// ---- Modules/12 FG_02/FG_02.TcPOU
// FG_02 - optical inspection. Camera handshake, no moving parts.
// Triggered by Index02; reports OperationDone. A NOK aborts (fault 1).
// Twin side: FB_Camera in OC_SIM - both halves must agree on the bit layout,
// and nothing checks it for you.
// Contract: _workflow/reference/fg-02-behaviour.md
FUNCTION_BLOCK FG_02 EXTENDS FB_PackML_BaseModule
VAR
	P_Camera	: FB_AbstractCamera := (Name := 'P_Camera');

	// Group level fault - see ST_FG_02_Inspection_Status. Cleared in Clearing.
	_FaultCode		: DINT;
	// The verdict of the last completed shot, latched so the panel still shows it
	// once ResultValid has dropped.
	_LastResultOK	: BOOL;

	{ attribute 'TcHmiSymbol.AddSymbol' }
	HMI : ST_HMI_FG_02;
END_VAR

METHOD PROTECTED Aborting
VAR_INPUT
END_VAR
// Disable() drops the trigger before the enable, so a shot is never left armed.
CASE SequenceState OF
	0:
		NoStateTasksToComplete	:= FALSE;
		P_Camera.Disable();
		SequenceState			:= SequenceState + 10;

	10:
		StateTasksComplete := TRUE;
END_CASE

SUPER^.Aborting();
END_METHOD

METHOD PROTECTED Clearing
VAR_INPUT
END_VAR
CASE SequenceState OF
	0:
		NoStateTasksToComplete := FALSE;
		// Cleared by the act of clearing, not by the condition going away.
		_FaultCode := 0;
		SequenceState := SequenceState + 10;

	10:	// Clear any latched component alarm.
		IF P_Camera.Reset() THEN
			SequenceState := SequenceState + 10;
		END_IF

	20:
		StateTasksComplete := TRUE;
END_CASE

SUPER^.Clearing();
END_METHOD

METHOD PUBLIC CyclicLogic
VAR_INPUT
END_VAR
IF NOT _InitComplete THEN
	_InitComplete := Initialize();
	RETURN;
END_IF

// No process image copy step: component members map straight to terminal channels.
SUPER^.CyclicLogic();

PublishStatus();
END_METHOD

METHOD PROTECTED Execute
VAR_INPUT
END_VAR
VAR_INST
	ReadyTimer	: TON;
	ShotTimer	: TON;
END_VAR
// The vision-sensor handshake. Every wait is bounded; every timeout faults.

CASE _CurrentMode OF

	//============================= PRODUCTION =================================
	E_PMLUnitMode.ePMLUnitMode_Production:

		CASE SequenceState OF
			0:
				NoStateTasksToComplete	:= FALSE;
				P_Camera.Disable();
				SequenceState			:= SequenceState + 10;

			10:	// Power up, wait for Ready. Timeout -> the camera is not answering.
				P_Camera.Enable();
				IF P_Camera.Ready THEN
					SequenceState := SequenceState + 10;
				ELSIF ReadyTimer.Q THEN
					_FaultCode := 2;
					AbortImmediate();
				END_IF

			20:	// Trigger. ResultValid also acknowledges: a fast camera can raise
				// and drop Busy inside one scan.
				P_Camera.Trigger();
				IF P_Camera.DeviceBusy OR P_Camera.ResultValid THEN
					SequenceState := SequenceState + 10;
				ELSIF ShotTimer.Q THEN
					_FaultCode := 3;
					AbortImmediate();
				END_IF

			30:	// Read the verdict. It stands until the trigger is released.
				IF P_Camera.ResultValid THEN
					_LastResultOK := P_Camera.ResultOK;
					IF P_Camera.ResultOK THEN
						SequenceState := SequenceState + 10;
					ELSE
						_FaultCode := 1;
						AbortImmediate();
					END_IF
				ELSIF ShotTimer.Q THEN
					_FaultCode := 3;
					AbortImmediate();
				END_IF

			40:	// Power down. Disable() clears the trigger first, which tells the
				// camera its verdict was read.
				P_Camera.Disable();
				SequenceState := SequenceState + 10;

			50:	// Execute is the one acting state that does not self-complete.
				// StateComplete() would be wrong here.
				ChangeState(E_PMLCommand.ePMLCommand_Complete);
		END_CASE

	//======================= MAINTENANCE & MANUAL =============================
	E_PMLUnitMode.ePMLUnitMode_Maintenance, E_PMLUnitMode.ePMLUnitMode_Manual:
		// No group sequence. The camera stays reachable through its own
		// component HMI control.
		;
END_CASE

SUPER^.Execute();

// ShotTimer spans steps 20 and 30 on purpose: the camera's total response time is
// one number, and that is what an operator is told.
ReadyTimer(IN := SequenceState = 10,								PT := T#2S);
ShotTimer(IN := (SequenceState = 20) OR (SequenceState = 30),		PT := T#3S);
END_METHOD

METHOD PROTECTED HMICommunication
VAR_INPUT
END_VAR
// Command half of the HMI bridge; PublishStatus is the status half. MUST be in
// this method: the base calls it immediately before ModeControl() and
// StateControl(), and reads its own PackMLBaseModule_HMI.Command, never ours.
PackMLBaseModule_HMI.Command := HMI.Command;

SUPER^.HMICommunication();

// The base clears a latch by writing back the value it acted on.
HMI.Command := PackMLBaseModule_HMI.Command;
END_METHOD

METHOD PROTECTED Initialize : BOOL;
VAR
END_VAR
Initialize := FALSE;

CASE DescendantSequenceState OF
	0:
		RegisterComponent(P_Camera);

		_LogModeChanges		:= FALSE;
		_LogStateChanges	:= TRUE;
		HMI.Config.Name		:= THIS^._Name;
		DescendantSequenceState := DescendantSequenceState + 10;

	10:
		// No travel timeouts - nothing in this group moves.
		DescendantSequenceState := DescendantSequenceState + 10;

	20:
		IF SUPER^.Initialize() THEN
			DescendantSequenceState := DescendantSequenceState + 10;
		END_IF

	30:
		Initialize := TRUE;
END_CASE
END_METHOD

ACTION PublishStatus:
// Status half of the HMI bridge. Called AFTER SUPER^.CyclicLogic(), so every
// field is this scan's. Copy the base struct wholesale - setting fields one by one
// leaves Busy, Error, ErrorID and HMIControlAvailable at zero.
// P_Camera publishes its own handshake; what is added here is what no device owns.
HMI.Config		:= PackMLBaseModule_HMI.Config;
HMI.Status		:= PackMLBaseModule_HMI.Status;

HMI.StateName				:= F_PMLStateName(_CurrentState);
HMI.Sequence.StepIndex		:= SequenceState;
HMI.Inspection.FaultCode	:= _FaultCode;
HMI.Inspection.LastResultOK	:= _LastResultOK;
END_ACTION

METHOD PROTECTED Resetting
VAR_INPUT
END_VAR
// Home is "nothing energised". Terminates on its own call and nothing else.

CASE SequenceState OF
	0:
		NoStateTasksToComplete	:= FALSE;
		P_Camera.Disable();
		SequenceState			:= SequenceState + 10;

	10:
		StateTasksComplete := TRUE;
END_CASE

SUPER^.Resetting();
END_METHOD

METHOD PROTECTED Stopping
VAR_INPUT
END_VAR
CASE SequenceState OF
	0:
		NoStateTasksToComplete	:= FALSE;
		P_Camera.Disable();
		SequenceState			:= SequenceState + 10;

	10:
		StateTasksComplete := TRUE;
END_CASE

SUPER^.Stopping();
END_METHOD

END_FUNCTION_BLOCK

// ---- Modules/13 FG_03/FG_03.TcPOU
// FG_03 - slot 1 to slot 2 transfer, with a 180 degree flip.
// !! THE TWO ARMS NAME THEIR AXES THE OPPOSITE WAY ROUND. Arm 1: X1 vertical,
// Y1 horizontal. Arm 2: X2 horizontal, Y2 vertical (factor -0.001, so a rising
// value descends). Every earlier version of this file had arm 1 wrong.
// Arm 1 NEVER lowers to place - the R1 flip is what carries the part down.
// A cylinder limit is not a grip witness: only B_Detect1/B_Detect2 are.
// Contract: _workflow/reference/fg-03-behaviour.md and gripper-station-reset.md
FUNCTION_BLOCK FG_03 EXTENDS FB_PackML_BaseModule
VAR
	// --- Arm 1, the placing arm ---------------------------------------------
	{ attribute 'TcHmiSymbol.AddSymbol' }
	Y_AxisX1	: FB_DoubleSolenoidFeedback := (Name := 'Y_AxisX1');
	{ attribute 'TcHmiSymbol.AddSymbol' }
	Y_AxisY1	: FB_DoubleSolenoidFeedback := (Name := 'Y_AxisY1');
	{ attribute 'TcHmiSymbol.AddSymbol' }
	Y_AxisR1	: FB_DoubleSolenoidFeedback := (Name := 'Y_AxisR1');
	{ attribute 'TcHmiSymbol.AddSymbol' }
	Y_Gripper1	: FB_DoubleSolenoidFeedback := (Name := 'Y_Gripper1');
	{ attribute 'TcHmiSymbol.AddSymbol' }
	B_Detect1	: FB_DigitalSensor := (Name := 'B_Detect1');

	// --- Arm 2, the picking arm ---------------------------------------------
	{ attribute 'TcHmiSymbol.AddSymbol' }
	Y_AxisX2	: FB_DoubleSolenoidFeedback := (Name := 'Y_AxisX2');
	{ attribute 'TcHmiSymbol.AddSymbol' }
	Y_AxisY2	: FB_DoubleSolenoidFeedback := (Name := 'Y_AxisY2');
	{ attribute 'TcHmiSymbol.AddSymbol' }
	Y_Gripper2	: FB_DoubleSolenoidFeedback := (Name := 'Y_Gripper2');
	{ attribute 'TcHmiSymbol.AddSymbol' }
	B_Detect2	: FB_DigitalSensor := (Name := 'B_Detect2');

	// Group level fault - see ST_FG_03_Transfer_Status. Cleared in Clearing.
	_FaultCode	: DINT;

	// What Resetting found in the grippers, sampled ONCE at its step 0. They decide
	// which grippers it may open and which way it turns arm 1, and the fact that they
	// are a snapshot rather than a live read is the whole reason the reset cannot
	// hang: no step waits on a sensor, only on its own cylinders. Step 10 clears
	// _Held2 when it has VERIFIED arm 2 let go - updating the snapshot from a checked
	// fact, which is not the same thing as reading the sensor in a wait.
	_Held1		: BOOL;
	_Held2		: BOOL;

	{ attribute 'TcHmiSymbol.AddSymbol' }
	HMI : ST_HMI_FG_03;
END_VAR

METHOD PROTECTED Aborting
VAR_INPUT
END_VAR
// AN ABORT COMMANDS NO MOTION IN THIS GROUP, and that is the whole design.
// No hazardous output to kill. What there is, at almost every step, is a part held
// in the air, and commanding an axis on an abort risks dropping it.
// COMMANDING NOTHING IS NOT THE SAME AS HOLDING ON: the grippers are held closed
// by the CyclicLogic interlock. This method leaves the AXES alone.
// Homing happens in Resetting, where the operator has asked for it.
CASE SequenceState OF
	0:
		NoStateTasksToComplete	:= FALSE;
		SequenceState			:= SequenceState + 10;

	10:
		StateTasksComplete := TRUE;
END_CASE

SUPER^.Aborting();
END_METHOD

METHOD PROTECTED Clearing
VAR_INPUT
END_VAR
CASE SequenceState OF
	0:
		NoStateTasksToComplete := FALSE;
		// The group fault is cleared by the act of clearing, not by the condition
		// going away. A part jammed in a gripper is still jammed after the sensor
		// has stopped being interesting; the operator has to have taken it out, and
		// Execute's step 0 guard is what checks that they did.
		_FaultCode := 0;
		SequenceState := SequenceState + 10;

	10:	// Clear latched component alarms - the solenoid travel timeouts latch.
		IF Y_AxisX1.Reset()
			AND Y_AxisY1.Reset()
			AND Y_AxisR1.Reset()
			AND Y_Gripper1.Reset()
			AND B_Detect1.Reset()
			AND Y_AxisX2.Reset()
			AND Y_AxisY2.Reset()
			AND Y_Gripper2.Reset()
			AND B_Detect2.Reset() THEN
			SequenceState := SequenceState + 10;
		END_IF

	20:
		StateTasksComplete := TRUE;
END_CASE

SUPER^.Clearing();
END_METHOD

METHOD PUBLIC CyclicLogic
VAR_INPUT
END_VAR
IF NOT _InitComplete THEN
	_InitComplete := Initialize();
	RETURN;
END_IF

// A HELD PART IS GRIPPED ACTIVELY, IN EVERY STATE EXCEPT Execute.
//
// A DE-ENERGISED DOUBLE SOLENOID DOES NOT HOLD THE PART IN THE TWIN. True of the
// real valve, false here. The scene wires the gripper cylinder as:
//     OnLimitMaxEvent  -> Gripper.Pick(bool)
//     OnLimitMinEvent  -> Gripper.Place(bool)
//     OnActiveChanged  -> Gripper.Place(bool)    IsActive = "moving"
// and Cylinder sets IsActive := (target <> value), so the payload is held only
// while the cylinder is at max AND STANDING STILL. Leaving it uncommanded through
// Clearing and Resetting was enough to nudge it off the limit, and arm 1 dropped
// its part mid-reset.
//
// So the grip is re-asserted every scan off the live sensor. It commands no MOTION
// - Extend on a closed gripper is a no-op at the valve.
// BEFORE SUPER^, WHICH IS WHAT MAKES IT AN INTERLOCK: it overwrites whatever a
// state method asked for on the previous scan. HMICommunication runs inside SUPER^
// and still gets the last word, so Manual can jog a gripper open.
// Execute is excluded because Execute is the only state allowed to put a part down.
IF _CurrentState <> E_PMLState.ePMLState_Execute THEN
	IF B_Detect1.Active THEN
		Y_Gripper1.Extend();
	END_IF
	IF B_Detect2.Active THEN
		Y_Gripper2.Extend();
	END_IF
END_IF

// No process image copy step: component process-image members are mapped directly
// to terminal channels.
SUPER^.CyclicLogic();

PublishStatus();
END_METHOD

METHOD PROTECTED Execute
VAR_INPUT
END_VAR
VAR_INST
	SettleTimer		: TON;

	// One grace timer per confirming step, and they cannot be shared. Steps 90 and
	// 100 are adjacent, so a timer armed on "either of them" would never see its IN
	// drop between the two and would carry step 80's elapsed time into step 90.
	// Each is armed only once its cylinder has reached its limit: the cylinder's own
	// ExtendTime/RetractTime covers the travel, and this covers only the question
	// that follows it - did the payload do what the stroke was supposed to make it do.
	PickTimer		: TON;
	HandoverTimer	: TON;
	Release2Timer	: TON;
	Release1Timer	: TON;
END_VAR
// Ordering from the authored Process entry, confirmed motion by motion against
// The SIL's 0.2 s dwells are replaced by the limit switches they stood in for.
// EVERY GRIP AND EVERY RELEASE IS CONFIRMED BY A SENSOR, not by the cylinder limit
// alone: a gripper closing on nothing reaches Extended SOONER than one closing on
// a part, so .Extended proves the jaws moved, never that they caught anything.
// Each confirmation is bounded and faults rather than waiting; the cylinder's own
// travel timeout covers the stroke, these timers only the question after it.

CASE _CurrentMode OF

	//============================= PRODUCTION =================================
	E_PMLUnitMode.ePMLUnitMode_Production:

		CASE SequenceState OF
			0:	// WHERE THE CYCLE STARTS IS DERIVED, NOT REMEMBERED. A part in a
				// gripper is a legal starting condition: Resetting parks a held part
				// at its arm's safe position instead of putting it back, so the next
				// Start picks the cycle up from there. Which sub-sequence that is
				// follows from which gripper is carrying something and from nothing
				// else - no stored step index, no "was I interrupted" flag.
				//
				// The arm must actually BE at its safe position. If a part is held
				// somewhere else - someone jogged an axis in Manual - the entry point
				// would be a guess, so this refuses rather than moves. Reset is the
				// recovery: Resetting reaches a safe position from anywhere.
				NoStateTasksToComplete	:= FALSE;

				IF B_Detect1.Active THEN
					IF Y_AxisX1.Extended AND Y_AxisY1.Retracted AND Y_AxisR1.Retracted THEN
						SequenceState := 100;		// at SAFE B - resume into SUB 3
					ELSE
						_FaultCode := 5;
						AbortImmediate();
					END_IF

				ELSIF B_Detect2.Active THEN
					IF Y_AxisX2.Retracted AND Y_AxisY2.Retracted THEN
						SequenceState := 50;		// at SAFE A - resume into SUB 2
					ELSE
						_FaultCode := 5;
						AbortImmediate();
					END_IF

				ELSE
					SequenceState := 10;			// nothing held - the whole cycle
				END_IF

			10:	// Let the pallet settle on the index lift before touching it. No
				// sensor reports this, so it is a timer. A resume skips this step
				// entirely - the pallet has been standing still since the E-Stop.
				IF SettleTimer.Q THEN
					SequenceState := SequenceState + 10;
				END_IF

		//===================== SUB 1 - pick out of slot 1 ======================
		// Entered only with both grippers empty. Ends at SAFE A.
			20:	// Arm 2 down into slot 1. Arm in Ready pos
				Y_AxisX1.Extend();
				Y_AxisY2.Extend();
				IF Y_AxisY2.Extended THEN
					SequenceState := SequenceState + 10;
				END_IF
				

			30:	// Grip the part, and confirm the grip caught something. An empty
				// slot 1, a mispositioned pallet or a part that slipped all look
				// identical on the cylinder limit and are all fault 2 here.
				Y_Gripper2.Extend();
				IF Y_Gripper2.Extended THEN
					IF B_Detect2.Active THEN
						SequenceState := SequenceState + 10;
					ELSIF PickTimer.Q THEN
						_FaultCode := 2;
						AbortImmediate();
					END_IF
				END_IF

			40:	// Lift clear of the pallet before anything traverses.
				//
				// *** SAFE A *** - X2 min, Y2 min, part in gripper 2. Arm 2 raised at
				// its home over slot 1. This is a state the cycle passes through in
				// the ordinary course, which is why a resume re-enters at step 50 and
				// nothing had to be inserted to make the position real.
				Y_AxisY2.Retract();
				IF Y_AxisY2.Retracted THEN
					SequenceState := SequenceState + 10;
				END_IF

		//=================== SUB 2 - the transfer (resume: 50) =================
		// Entered with the part in gripper 2 and arm 2 at SAFE A. Ends at SAFE B.
			50:	// Arm 2 traverses to the transfer position
				Y_AxisX2.Extend();
				IF Y_AxisX2.Extended THEN
					SequenceState := SequenceState + 10;
				END_IF

			60:	// ARM 1 RISES, AND THEN STAYS UP FOR THE WHOLE CYCLE. 			
				IF Y_AxisX1.Extended THEN
					SequenceState := SequenceState + 10;
				END_IF

			70:	// Arm 1 traverses across to meet arm 2. 
				Y_AxisY1.Extend();
				IF Y_AxisY1.Extended THEN
					SequenceState := SequenceState + 10;
				END_IF

			80:	// Arm 1 takes hold. BOTH GRIPPERS NOW HOLD THE PART, and what makes
				// the next step safe is B_Detect1 - not the cylinder limit. Arm 1's
				// jaws reach Extended whether or not the part is between them, and a
				// dwell here (which is what the SIL does) proves even less. Only the
				// sensor says arm 1 actually has it, and step 90 opens arm 2 on the
				// strength of that.
				//
				// THIS IS THE ONE WINDOW WITH NO SAFE POSITION. Neither arm can move
				// while both hold one part, which is why Resetting has to break the
				// tie here before it can park anything.
				Y_Gripper1.Extend();
				IF Y_Gripper1.Extended THEN
					IF B_Detect1.Active THEN
						SequenceState := SequenceState + 10;
					ELSIF HandoverTimer.Q THEN
						_FaultCode := 3;
						AbortImmediate();
					END_IF
				END_IF

			90:	// Arm 2 lets go. Only now, and only once the part has actually left
				// its jaws - a part still in the beam when arm 2 traverses away would
				// be dragged off arm 1.
				//
				// *** SAFE B *** - X1 max, Y1 max, R1 min, part in gripper 1. Arm 1
				// raised at the transfer position, holding the part unrotated. Like
				// SAFE A this is a state the cycle really passes through, so a resume
				// re-enters at step 100 and simply carries on.
				Y_Gripper2.Retract();
				IF Y_Gripper2.Retracted THEN
					IF NOT B_Detect2.Active THEN
						SequenceState := SequenceState + 10;
					ELSIF Release2Timer.Q THEN
						_FaultCode := 4;
						AbortImmediate();
					END_IF
				END_IF

		//================= SUB 3 - place into slot 2 (resume: 100) =============
		// Entered with the part in gripper 1 at SAFE B.
			100: // Arm 2 back home over slot 1, empty. 
				Y_AxisX2.Retract();
				IF Y_AxisX2.Retracted THEN
					SequenceState := 105;
				END_IF
				
			105: //Align arm 1 with slot
				Y_AxisY1.Extend();
				IF Y_AxisY1.Extended THEN
					SequenceState := 110;
				END_IF

			110: // THE FLIP, AND IT IS ALSO THE PLACING MOVE. 
				Y_AxisR1.Extend();
				IF Y_AxisR1.Extended THEN
					SequenceState := SequenceState + 10;
				END_IF

			120: // Traverse across to slot 2, carrying the part flipped
				Y_AxisX1.Retract();
				IF Y_AxisX1.Retracted THEN
					SequenceState := SequenceState + 10;
				END_IF

			130: // Release into slot 2. Confirm the part is out of the jaws before
				// arm 1 traverses away: a part still gripped is carried back out of
				// the pallet, and Index03 would release a pallet that looks finished
				// and is empty.
				Y_Gripper1.Retract();
				IF Y_Gripper1.Retracted THEN
					IF NOT B_Detect1.Active THEN
						SequenceState := SequenceState + 10;
					ELSIF Release1Timer.Q THEN
						_FaultCode := 4;
						AbortImmediate();
					END_IF
				END_IF

			140: // Traverse clear of the part just placed. THIS IS NOT A DETOUR: the
				// rotation home at step 150 sweeps the gripper through wherever it
				// stands, and over slot 2 that is straight through the part. Arm 1
				// has to be back at the transfer position before it may turn.
				Y_AxisX1.Extend();
				IF Y_AxisX1.Extended THEN
					SequenceState := SequenceState + 10;
				END_IF

			150: // Rotate home, empty and clear
				Y_AxisR1.Retract();
				IF Y_AxisR1.Retracted THEN
					SequenceState := SequenceState + 10;
				END_IF

			160: // And back to the home position over slot 2
				Y_AxisY1.Retract();
				IF Y_AxisY1.Retracted THEN
					SequenceState := SequenceState + 10;
				END_IF

			170: // Execute is the one acting state that does not self-complete.
				// StateComplete() would be wrong here.
				ChangeState(E_PMLCommand.ePMLCommand_Complete);
		END_CASE

	//======================= MAINTENANCE & MANUAL =============================
	E_PMLUnitMode.ePMLUnitMode_Maintenance, E_PMLUnitMode.ePMLUnitMode_Manual:
		// Every cylinder is jogged through its own SolenoidHMI command struct,
		// which FB_SingleSolenoid.HMICommunication honours whenever HMIPermissions
		// has granted control. No group sequence runs and no code is needed here.
		;
END_CASE

SUPER^.Execute();

SettleTimer(IN := SequenceState = 10, PT := T#500MS);

// The payload grace timers. Each is armed only once its cylinder has reached the
// limit, so the budget is for the part settling in or falling out of the jaws, not
// for the stroke - the stroke already has ExtendTime/RetractTime on the cylinder.
// 500 ms is generous for a beam sensor that answers within one twin frame; it is
// long enough that a slow physics step cannot fault a good grip.
PickTimer(IN		:= (SequenceState = 30)  AND Y_Gripper2.Extended,	PT := T#500MS);
HandoverTimer(IN	:= (SequenceState = 80)  AND Y_Gripper1.Extended,	PT := T#500MS);
Release2Timer(IN	:= (SequenceState = 90)  AND Y_Gripper2.Retracted,	PT := T#500MS);
Release1Timer(IN	:= (SequenceState = 130) AND Y_Gripper1.Retracted,	PT := T#500MS);
END_METHOD

METHOD PROTECTED HMICommunication
VAR_INPUT
END_VAR
// The command half of the HMI bridge; PublishStatus is the status half.
//
// The base reads its OWN PackMLBaseModule_HMI.Command and never looks at ours, so
// without this a mode or state button on the FG_03 tile writes into a struct
// nothing consumes. It has to happen in this method because the base calls it
// immediately before ModeControl() and StateControl().
PackMLBaseModule_HMI.Command := HMI.Command;

SUPER^.HMICommunication();

// The base clears a latch by writing back the value it acted on, so the panel
// sees its request consumed instead of re-issuing it next scan.
HMI.Command := PackMLBaseModule_HMI.Command;
END_METHOD

METHOD PROTECTED Initialize : BOOL;
VAR
END_VAR
Initialize := FALSE;

CASE DescendantSequenceState OF
	0:
		RegisterComponent(Y_AxisX1);
		RegisterComponent(Y_AxisY1);
		RegisterComponent(Y_AxisR1);
		RegisterComponent(Y_Gripper1);
		RegisterComponent(B_Detect1);
		RegisterComponent(Y_AxisX2);
		RegisterComponent(Y_AxisY2);
		RegisterComponent(Y_Gripper2);
		RegisterComponent(B_Detect2);

		_LogModeChanges		:= FALSE;
		_LogStateChanges	:= TRUE;
		HMI.Config.Name		:= THIS^._Name;
		DescendantSequenceState := DescendantSequenceState + 10;

	10:
		// Travel timeouts in ms (LREAL). The twin completes a stroke well inside
		// these; they exist to alarm on a jam, not to pace the cycle. Allowed by
		// ROLE, not by name: the horizontal traverses and the rotate get the long
		// budget, the vertical strokes and the grippers the short one - and on arm
		// 1 it is X1 that is vertical and Y1 that traverses.
		Y_AxisX1.ExtendTime			:= 2000.0;	// vertical
		Y_AxisX1.RetractTime		:= 2000.0;
		Y_AxisY1.ExtendTime			:= 3000.0;	// horizontal traverse
		Y_AxisY1.RetractTime		:= 3000.0;
		Y_AxisR1.ExtendTime			:= 3000.0;
		Y_AxisR1.RetractTime		:= 3000.0;
		Y_Gripper1.ExtendTime		:= 2000.0;
		Y_Gripper1.RetractTime		:= 2000.0;
		Y_AxisX2.ExtendTime			:= 3000.0;
		Y_AxisX2.RetractTime		:= 3000.0;
		Y_AxisY2.ExtendTime			:= 2000.0;
		Y_AxisY2.RetractTime		:= 2000.0;
		Y_Gripper2.ExtendTime		:= 2000.0;
		Y_Gripper2.RetractTime		:= 2000.0;
		DescendantSequenceState := DescendantSequenceState + 10;

	20:
		IF SUPER^.Initialize() THEN
			DescendantSequenceState := DescendantSequenceState + 10;
		END_IF

	30:
		Initialize := TRUE;
END_CASE
END_METHOD

ACTION PublishStatus:
// Local HMI surface, and the status half of the HMI bridge - HMICommunication is
// the command half. Called from CyclicLogic AFTER SUPER^.CyclicLogic(), so every
// field is this scan's. Copy the base struct wholesale - setting fields one by
// one leaves Busy, Error, ErrorID and HMIControlAvailable at zero.
// Every device publishes itself; what is added here is what no device owns.
//
// ResumePoint IS DERIVED HERE, NOT COPIED FROM _Held1/_Held2. Those are Resetting's
// private snapshot and are stale everywhere else. This runs the same derivation
// Execute step 0 runs, off the live sensors, so the panel shows what pressing Start
// would actually do.
HMI.Config		:= PackMLBaseModule_HMI.Config;
HMI.Status		:= PackMLBaseModule_HMI.Status;

HMI.StateName				:= F_PMLStateName(_CurrentState);
HMI.Sequence.StepIndex		:= SequenceState;
HMI.Transfer.FaultCode		:= _FaultCode;

IF B_Detect1.Active THEN
	HMI.Transfer.ResumePoint := 3;		// place into slot 2
ELSIF B_Detect2.Active THEN
	HMI.Transfer.ResumePoint := 2;		// the handover
ELSE
	HMI.Transfer.ResumePoint := 1;		// the whole cycle
END_IF
END_ACTION

METHOD PROTECTED Resetting
VAR_INPUT
END_VAR
// Bring both arms to their SAFE POSITIONS, keeping hold of whatever they are
// holding. This state does not undo the cycle and does not finish it - it puts the
// machine somewhere Execute step 0 can pick up again.
//
// THE SAFE POSITIONS ARE STATES THE CYCLE ALREADY RESTS AT - neither was invented:
//   SAFE A   X2 min, Y2 min          arm 2 raised at home over slot 1, holding.
//                                    Left by step 40; resume at step 50.
//   SAFE B   X1 max, Y1 max, R1 min  arm 1 raised at the TRANSFER position,
//                                    holding, not yet rotated. Left by step 90;
//                                    resume at step 100.
// Arm 1's safe position is NOT its home: home is Y1 min over slot 2, the place
// position, where a part would hover un-rotated and wrong way up.
//
// THE GRIPPERS ARE HELD CLOSED, NOT LEFT ALONE - see CyclicLogic. Only empty
// grippers are driven open.
//
// THE SENSORS ARE SAMPLED ONCE, AT STEP 0, AND NEVER READ AGAIN. From then on every
// step waits on its own cylinders and nothing else - not a sensor, not another
// unit, not an event that may not arrive. A snapshot cannot fail to arrive.
//
// STEPS 80..90 ARE THE ONE WINDOW WITH NO SAFE POSITION: both grippers hold the
// same part and moving either arm tears it. Step 10 below is entered only for that
// case. ARM 1 HAS PRIORITY - it keeps the part, arm 2 lets go, resume from SAFE B.

CASE SequenceState OF
	0:
		NoStateTasksToComplete	:= FALSE;

		_Held1 := B_Detect1.Active;
		_Held2 := B_Detect2.Active;

		IF _Held1 AND _Held2 THEN
			SequenceState := 10;
		ELSE
			SequenceState := 100;
		END_IF

	//============ 10 - both grippers hold one part, mid-transfer ==============
	10:	// Arm 1 has priority, so arm 2 is the one that lets go - which is also
		// exactly what Execute step 90 does, at the position the arms already
		// stand in, before anything travels.
		Y_Gripper2.Retract();
		IF Y_Gripper2.Retracted THEN
			IF B_Detect2.Active THEN
				// ARM 2 HAS NOT LET GO, SO NOTHING MOVES. Every path from here
				// separates the arms, and separating them while both still hold
				// the part is the failure this method exists to remove. The reset
				// completes where it stands - arms at the transfer, part held,
				// code 1 raised - and Execute's step 0 refuses the next cycle
				// because the part is not at a safe position. Terminating on time
				// without moving is the safe answer; parking at any cost is not.
				_FaultCode		:= 1;
				SequenceState	:= 900;
			ELSE
				_Held2			:= FALSE;	// verified empty, not assumed
				SequenceState	:= 100;
			END_IF
		END_IF

	//================== 100 - to the safe positions ===========================
	100: //Arm 2 to home
		Y_AxisX2.Retract();
		Y_AxisY2.Retract();
		IF Y_AxisX2.Retracted AND Y_AxisY2.Retracted THEN
			SequenceState := SequenceState + 10;
		END_IF

	110: //ARm 1 to home
		Y_AxisX1.Extend();
		Y_AxisY1.Retract();
		
		IF Y_AxisX1.Extended AND Y_AxisY1.Retracted THEN
			SequenceState := SequenceState + 10;
		END_IF

	120: // Rotate home. ONLY EVER HERE: over slot 2 the sweep goes straight
		// through whatever is in the slot, which is why Execute traverses back to
		// this position at step 140 before turning at 150. Turning with a part
		// held is Execute step 110's move, so it is safe loaded too.
		Y_AxisR1.Retract();
		IF Y_AxisR1.Retracted THEN
			SequenceState := SequenceState + 10;
		END_IF

	130: // Open the EMPTY grippers, and only those. A gripper holding a part is
		// not touched here - CyclicLogic is holding it closed, and that command
		// wins because it runs first. The wait is on the cylinders this step
		// actually commanded: a held gripper contributes no condition, because
		// there is nothing to wait for.
		IF NOT _Held1 THEN
			Y_Gripper1.Retract();
		END_IF
		IF NOT _Held2 THEN
			Y_Gripper2.Retract();
		END_IF

		IF (_Held1 OR Y_Gripper1.Retracted) AND (_Held2 OR Y_Gripper2.Retracted) THEN
			SequenceState := 900;
		END_IF

	//========================== common exit ===================================
	900:
		StateTasksComplete := TRUE;
END_CASE

SUPER^.Resetting();
END_METHOD

METHOD PROTECTED Stopping
VAR_INPUT
END_VAR
// A controlled stop commands no axis motion, for the same reason an abort does not:
// the part is held in the air for most of this cycle. The grip itself is held by
// the CyclicLogic interlock, not by leaving the valve alone. The transfer is
// resumed by a reset, which parks the part at a safe position.
CASE SequenceState OF
	0:
		NoStateTasksToComplete	:= FALSE;
		SequenceState			:= SequenceState + 10;

	10:
		StateTasksComplete := TRUE;
END_CASE

SUPER^.Stopping();
END_METHOD

END_FUNCTION_BLOCK

// ---- Modules/14 FG_04/FG_04.TcPOU
// FG_04 - press and seat check. Y_AxisZ (double solenoid) and B_NIO.
// Triggered by Index04; reports OperationDone. An NIO aborts (fault 1).
// B_NIO IS A VERDICT, NOT A SENSOR READING: the twin's PartPressDetector raises
// it only at the bottom limit with the hold expired, so step 30 is the one place
// it means anything. Contract: _workflow/reference/fg-04-behaviour.md
FUNCTION_BLOCK FG_04 EXTENDS FB_PackML_BaseModule
VAR
	{ attribute 'TcHmiSymbol.AddSymbol' }
	Y_AxisZ		: FB_DoubleSolenoidFeedback := (Name := 'Y_AxisZ');
	{ attribute 'TcHmiSymbol.AddSymbol' }
	B_NIO		: FB_DigitalSensor := (Name := 'B_NIO');

	// Group level fault. One code - see ST_FG_04_Press_Status. Cleared in Clearing.
	_FaultCode	: DINT;

	{ attribute 'TcHmiSymbol.AddSymbol' }
	HMI : ST_HMI_FG_04;
END_VAR

METHOD PROTECTED Aborting
VAR_INPUT
END_VAR
// LIFT THE PRESS - not a no-motion abort. A press held on a part is this
// station's hazardous state. Bounded by Y_AxisZ.RetractTime, so a jammed press
// alarms out of this state instead of parking in it.
CASE SequenceState OF
	0:
		NoStateTasksToComplete	:= FALSE;
		SequenceState			:= SequenceState + 10;

	10:
		Y_AxisZ.Retract();
		IF Y_AxisZ.Retracted THEN
			SequenceState := SequenceState + 10;
		END_IF

	20:
		StateTasksComplete := TRUE;
END_CASE

SUPER^.Aborting();
END_METHOD

METHOD PROTECTED Clearing
VAR_INPUT
END_VAR
CASE SequenceState OF
	0:
		NoStateTasksToComplete := FALSE;
		// Cleared by the act of clearing, not by the condition going away.
		_FaultCode := 0;
		SequenceState := SequenceState + 10;

	10:	// Clear latched component alarms - the solenoid travel timeouts latch.
		IF Y_AxisZ.Reset()
			AND B_NIO.Reset() THEN
			SequenceState := SequenceState + 10;
		END_IF

	20:
		StateTasksComplete := TRUE;
END_CASE

SUPER^.Clearing();
END_METHOD

METHOD PUBLIC CyclicLogic
VAR_INPUT
END_VAR
IF NOT _InitComplete THEN
	_InitComplete := Initialize();
	RETURN;
END_IF

// No process image copy step: component members map straight to terminal channels.
SUPER^.CyclicLogic();

PublishStatus();
END_METHOD

METHOD PROTECTED Execute
VAR_INPUT
END_VAR
VAR_INST
	SettleTimer	: TON;
	HoldTimer	: TON;
END_VAR
// settle 0.5 s -> press down -> hold 1 s -> read verdict -> retract.
// The hold is a timer because nothing reports "seated" - only B_NIO reports
// the opposite.

CASE _CurrentMode OF

	//============================= PRODUCTION =================================
	E_PMLUnitMode.ePMLUnitMode_Production:

		CASE SequenceState OF
			0:
				NoStateTasksToComplete	:= FALSE;
				SequenceState			:= SequenceState + 10;

			10:	// Let the pallet settle on the index lift before pressing on it
				IF SettleTimer.Q THEN
					SequenceState := SequenceState + 10;
				END_IF

			20:	// Down onto the part
				Y_AxisZ.Extend();
				IF Y_AxisZ.Extended THEN
					SequenceState := SequenceState + 10;
				END_IF

			30:	// Hold at the bottom, THEN read. B_NIO is only meaningful once the
				// press is at its limit and the hold has expired.
				IF HoldTimer.Q THEN
					IF B_NIO.Active THEN
						_FaultCode := 1;
						AbortImmediate();
					ELSE
						SequenceState := SequenceState + 10;
					END_IF
				END_IF

			40:	// Lift clear before the index lowers the pallet
				Y_AxisZ.Retract();
				IF Y_AxisZ.Retracted THEN
					SequenceState := SequenceState + 10;
				END_IF

			50:	// Execute is the one acting state that does not self-complete.
				// StateComplete() would be wrong here.
				ChangeState(E_PMLCommand.ePMLCommand_Complete);
		END_CASE

	//======================= MAINTENANCE & MANUAL =============================
	E_PMLUnitMode.ePMLUnitMode_Maintenance, E_PMLUnitMode.ePMLUnitMode_Manual:
		// No group sequence. Y_AxisZ stays jogged through its own component
			// HMI control.
		;
END_CASE

SUPER^.Execute();

SettleTimer(IN := SequenceState = 10,							PT := T#500MS);
HoldTimer(IN := (SequenceState = 30) AND Y_AxisZ.Extended,		PT := T#1S);
END_METHOD

METHOD PROTECTED HMICommunication
VAR_INPUT
END_VAR
// Command half of the HMI bridge; PublishStatus is the status half. MUST be in
// this method: the base calls it immediately before ModeControl() and
// StateControl(), and reads its own PackMLBaseModule_HMI.Command, never ours.
PackMLBaseModule_HMI.Command := HMI.Command;

SUPER^.HMICommunication();

// The base clears a latch by writing back the value it acted on.
HMI.Command := PackMLBaseModule_HMI.Command;
END_METHOD

METHOD PROTECTED Initialize : BOOL;
VAR
END_VAR
Initialize := FALSE;

CASE DescendantSequenceState OF
	0:
		RegisterComponent(Y_AxisZ);
		RegisterComponent(B_NIO);

		_LogModeChanges		:= FALSE;
		_LogStateChanges	:= TRUE;
		HMI.Config.Name		:= THIS^._Name;
		DescendantSequenceState := DescendantSequenceState + 10;

	10:
		// Travel timeouts in ms. On a press, alarming on a jam is what they are for.
		Y_AxisZ.ExtendTime	:= 2000.0;
		Y_AxisZ.RetractTime	:= 2000.0;
		DescendantSequenceState := DescendantSequenceState + 10;

	20:
		IF SUPER^.Initialize() THEN
			DescendantSequenceState := DescendantSequenceState + 10;
		END_IF

	30:
		Initialize := TRUE;
END_CASE
END_METHOD

ACTION PublishStatus:
// Status half of the HMI bridge. Called AFTER SUPER^.CyclicLogic(), so every
// field is this scan's. Copy the base struct wholesale - setting fields one by
// one leaves Busy, Error, ErrorID and HMIControlAvailable at zero.
HMI.Config		:= PackMLBaseModule_HMI.Config;
HMI.Status		:= PackMLBaseModule_HMI.Status;

HMI.StateName			:= F_PMLStateName(_CurrentState);
HMI.Sequence.StepIndex	:= SequenceState;
HMI.Press.FaultCode		:= _FaultCode;
END_ACTION

METHOD PROTECTED Resetting
VAR_INPUT
END_VAR
// Home is the press up. One cylinder, bounded by its own travel timeout.

CASE SequenceState OF
	0:
		NoStateTasksToComplete	:= FALSE;
		SequenceState			:= SequenceState + 10;

	10:
		Y_AxisZ.Retract();
		IF Y_AxisZ.Retracted THEN
			SequenceState := SequenceState + 10;
		END_IF

	20:
		StateTasksComplete := TRUE;
END_CASE

SUPER^.Resetting();
END_METHOD

METHOD PROTECTED Stopping
VAR_INPUT
END_VAR
// A stop lifts the press, for the same reason the abort does.
CASE SequenceState OF
	0:
		NoStateTasksToComplete	:= FALSE;
		SequenceState			:= SequenceState + 10;

	10:
		Y_AxisZ.Retract();
		IF Y_AxisZ.Retracted THEN
			SequenceState := SequenceState + 10;
		END_IF

	20:
		StateTasksComplete := TRUE;
END_CASE

SUPER^.Stopping();
END_METHOD

END_FUNCTION_BLOCK

// ---- Modules/15 FG_05/FG_05.TcPOU
// FG_05 - capping station.
// THE BUNKER IS NOT PART OF THE PALLET CYCLE. Y_CapsSource is commanded from
// CyclicLogic via DriveBunker, on mode and state only; driven from Execute it
// would stop between pallets and step 10 would block on B_Part for ever.
// B_Part is on the FEED (a cap has arrived); B_Detect is in the JAWS (this unit
// is carrying one). They are not interchangeable.
// Y_CapsSourceStopper is HELD, NEVER INDEXED: EXTENDED BLOCKS THE PATH, and the
// queue pushes the next cap against it as the gripper takes the one in front.
// Contract: _workflow/reference/fg-05-behaviour.md and gripper-station-reset.md
FUNCTION_BLOCK FG_05 EXTENDS FB_PackML_BaseModule
VAR
	// --- The cap handling unit ----------------------------------------------
	{ attribute 'TcHmiSymbol.AddSymbol' }
	Y_AxisX					: FB_DoubleSolenoidFeedback := (Name := 'Y_AxisX');
	{ attribute 'TcHmiSymbol.AddSymbol' }
	Y_AxisZ1				: FB_DoubleSolenoidFeedback := (Name := 'Y_AxisZ1');
	{ attribute 'TcHmiSymbol.AddSymbol' }
	Y_AxisZ2				: FB_DoubleSolenoidFeedback := (Name := 'Y_AxisZ2');
	{ attribute 'TcHmiSymbol.AddSymbol' }
	Y_AxisR					: FB_DoubleSolenoidFeedback := (Name := 'Y_AxisR');
	{ attribute 'TcHmiSymbol.AddSymbol' }
	Y_Gripper				: FB_DoubleSolenoidFeedback := (Name := 'Y_Gripper');
	{ attribute 'TcHmiSymbol.AddSymbol' }
	B_Detect				: FB_DigitalSensor := (Name := 'B_Detect');

	// --- The cap feed --------------------------------------------------------
	{ attribute 'TcHmiSymbol.AddSymbol' }
	Y_CapsSourceStopper		: FB_DoubleSolenoidFeedback := (Name := 'Y_CapsSourceStopper');
	Y_CapsSource			: FB_AbstractBunker := (Name := 'Y_CapsSource');
	{ attribute 'TcHmiSymbol.AddSymbol' }
	B_Part					: FB_DigitalSensor := (Name := 'B_Part');
	P_Camera				: FB_AbstractCamera := (Name := 'P_Camera');

	// Group level fault - see ST_FG_05_Capping_Status. Cleared in Clearing.
	_FaultCode				: DINT;
	// The verdict of the last completed read, latched so the panel still shows it
	// once ResultValid has dropped.
	_LastResultOK			: BOOL;
	// What Resetting found in the gripper, sampled ONCE at its step 0 and never
	// re-read. It decides which end of X the unit parks at and whether the reset
	// may open the gripper at all.
	_Held					: BOOL;

	{ attribute 'TcHmiSymbol.AddSymbol' }
	HMI : ST_HMI_FG_05;
END_VAR

METHOD PROTECTED Aborting
VAR_INPUT
END_VAR
// AN ABORT COMMANDS NO AXIS MOTION. For most of this cycle a cap is held in the air
// over the pallet. The grip is held by the CyclicLogic interlock, not by leaving
// the valve alone. Parking happens in Resetting, where the operator has asked for
// it.
//
// What does stop is everything that keeps running on its own: the feed, so caps
// stop arriving at a station that cannot take them, and the camera.
CASE SequenceState OF
	0:
		NoStateTasksToComplete	:= FALSE;
		Y_CapsSource.Halt();
		P_Camera.Disable();
		SequenceState			:= SequenceState + 10;

	10:
		StateTasksComplete := TRUE;
END_CASE

SUPER^.Aborting();
END_METHOD

METHOD PROTECTED Clearing
VAR_INPUT
END_VAR
CASE SequenceState OF
	0:
		NoStateTasksToComplete := FALSE;
		// The group fault is cleared by the act of clearing, not by the condition
		// going away - an assembly this station does not cap is still the wrong
		// assembly after the camera has stopped reporting it, and the operator has
		// to have dealt with the pallet.
		_FaultCode := 0;
		SequenceState := SequenceState + 10;

	10:	// Clear latched component alarms - the solenoid travel timeouts latch.
		IF Y_AxisX.Reset()
			AND Y_AxisZ1.Reset()
			AND Y_AxisZ2.Reset()
			AND Y_AxisR.Reset()
			AND Y_Gripper.Reset()
			AND B_Detect.Reset()
			AND Y_CapsSourceStopper.Reset()
			AND Y_CapsSource.Reset()
			AND B_Part.Reset()
			AND P_Camera.Reset() THEN
			SequenceState := SequenceState + 10;
		END_IF

	20:
		StateTasksComplete := TRUE;
END_CASE

SUPER^.Clearing();
END_METHOD

METHOD PUBLIC CyclicLogic
VAR_INPUT
END_VAR
IF NOT _InitComplete THEN
	_InitComplete := Initialize();
	RETURN;
END_IF

// The feed runs outside the pallet cycle - see the block header. Evaluated BEFORE
// the base walks its components so Y_CapsSource's own CyclicLogic publishes this
// scan's commanded state rather than last scan's, and so that in Manual mode its
// HMICommunication - which runs inside SUPER^ - still gets the last word on the
// output byte. That ordering is the whole reason an operator can jog the bunker.
DriveBunker();

// A HELD CAP IS GRIPPED ACTIVELY, IN EVERY STATE EXCEPT Execute. Identical
// interlock to FG_03's - a de-energised double solenoid does NOT hold the cap in
// the twin, because OnActiveChanged is wired to Gripper.Place and IsActive means
// MOVING. FG_03 dropped a part this way mid-reset; this station has the same
// wiring. Before SUPER^ so it overrides the state methods, while HMICommunication
// inside SUPER^ still lets Manual jog the gripper open.
IF _CurrentState <> E_PMLState.ePMLState_Execute THEN
	IF B_Detect.Active THEN
		Y_Gripper.Extend();
	END_IF
END_IF

// No process image copy step: component process-image members are mapped directly
// to terminal channels.
SUPER^.CyclicLogic();

PublishStatus();
END_METHOD

ACTION DriveBunker:
// The cap feed, which is not a step of anything.
//
// A BLACKLIST, NOT A WHITELIST, and deliberately: the feed should be running in
// every state where the station could plausibly be asked to work, and the states
// where it must not are few and nameable. Written the other way round, every
// PackML state anyone forgot would silently starve the pick position.
//
// Production only. In Maintenance and Manual the bunker belongs to the operator,
// through FB_AbstractBunker's own HMI command struct - the module keeps its hands
// off, and HMIPermissions has already granted control by the time SUPER^ runs.
IF _CurrentMode = E_PMLUnitMode.ePMLUnitMode_Production THEN

	CASE _CurrentState OF
		E_PMLState.ePMLState_Stopping,
		E_PMLState.ePMLState_Stopped,
		E_PMLState.ePMLState_Aborting,
		E_PMLState.ePMLState_Aborted,
		E_PMLState.ePMLState_Clearing:
			Y_CapsSource.Halt();
	ELSE
		Y_CapsSource.Run();
	END_CASE

ELSE
	Y_CapsSource.Halt();
END_IF
END_ACTION

METHOD PROTECTED Execute
VAR_INPUT
END_VAR
VAR_INST
	SettleTimer		: TON;
	ReadyTimer		: TON;
	ShotTimer		: TON;

	// One grace timer per payload confirmation, armed only once the gripper has
	// reached its limit. The cylinder's own ExtendTime/RetractTime covers the
	// stroke; these cover only the question that follows it.
	GripTimer		: TON;
	ReleaseTimer	: TON;
END_VAR
// Ordering from the authored Process entry. Every cylinder here is a *Feedback
// Both limits are wired, so the steps wait on limit switches, not dwells. The 0.5 s
// settle at step 10 is kept because no sensor reports it.
// Steps 20..50 are the vision-sensor protocol, identical to FG_01's and FG_02's,
// and every wait is bounded with a timeout raising a fault.
// AN ASSEMBLY THIS STATION DOES NOT CAP ABORTS THE GROUP; Index05 then raises its
// own fault 3 on the operation timeout. The abort is cheap only because the read is
// first - see the block header.
// These conditions name step numbers: renumbering a step moves its timer too.

CASE _CurrentMode OF

	//============================= PRODUCTION =================================
	E_PMLUnitMode.ePMLUnitMode_Production:

		CASE SequenceState OF
			0:	// WHERE THE CYCLE STARTS IS DERIVED, NOT REMEMBERED. A cap in the jaws
// is a legal starting condition: Resetting parks a held cap at the
				// SAFE POSITION, so the next Start picks the cycle up from there.
				// A RESUME SKIPS THE CAMERA, correctly: the read identifies the
				// ASSEMBLY, it ran before the pick and came back OK, and the pallet
				// has not moved. Re-reading asks a question already answered.
				// The unit must actually BE at the safe position - anywhere else the
				// entry point would be a guess, so this refuses rather than moves.
				NoStateTasksToComplete	:= FALSE;

				IF B_Detect.Active THEN
					IF Y_AxisX.Extended
						AND Y_AxisZ1.Retracted
						AND Y_AxisZ2.Retracted THEN
						SequenceState := 100;		// at SAFE - resume at the rotate
					ELSE
						_FaultCode := 4;
						AbortImmediate();
					END_IF
				ELSE
					P_Camera.Enable();
					P_Camera.ClearTrigger();
					SequenceState := SequenceState + 10;
				END_IF

			10:	// Nothing happens until there is a cap to pick. The stopper is EXTENDED
				// to block the path, so the queue accumulates against it; the feed
				// that fills it runs outside this sequence - see DriveBunker.
				Y_CapsSourceStopper.Extend();
				IF B_Part.Active AND SettleTimer.Q THEN
					SequenceState := SequenceState + 10;
				END_IF

			//--- Identify the assembly before picking a cap for it --------------
			20:	// Wait for the camera to say it can take a shot. It was enabled at
				// step 0 and step 10 has just spent at least 0.5 s waiting for a
				// cap, so Ready never arriving means the camera is not answering
				// at all - a wiring or device fault.
				IF P_Camera.Ready THEN
					SequenceState := SequenceState + 10;
				ELSIF ReadyTimer.Q THEN
					_FaultCode := 2;
					AbortImmediate();
				END_IF

			30:	// Ask for the shot. Busy is the acknowledgement, but a fast camera
				// can come and go inside one scan, so ResultValid counts as an
				// acknowledgement too - waiting only on Busy would hang on exactly
				// the device that answered quickest.
				P_Camera.Trigger();
				IF P_Camera.DeviceBusy OR P_Camera.ResultValid THEN
					SequenceState := SequenceState + 10;
				ELSIF ShotTimer.Q THEN
					_FaultCode := 3;
					AbortImmediate();
				END_IF

			40:	// Read the verdict. It stands until the trigger is released, so
				// this cannot miss it by being a scan late.
				IF P_Camera.ResultValid THEN
					_LastResultOK := P_Camera.ResultOK;
					IF P_Camera.ResultOK THEN
						SequenceState := SequenceState + 10;
					ELSE
						_FaultCode := 1;
						AbortImmediate();
					END_IF
				ELSIF ShotTimer.Q THEN
					_FaultCode := 3;
					AbortImmediate();
				END_IF

			50:	// Release the trigger. That is also what tells the camera its
				// verdict has been read, so it drops ResultValid and re-arms. The
				// enable stays on until the end of the cycle.
				P_Camera.ClearTrigger();
				SequenceState := SequenceState + 10;

			//--- Pick a cap off the feed ---------------------------------------
			60:	// Down on the bunker side
				Y_AxisZ2.Extend();
				IF Y_AxisZ2.Extended THEN
					SequenceState := SequenceState + 10;
				END_IF

			70:	// Grip the cap, and confirm the jaws caught it. B_Part said a cap
				// was AT the pick position; only B_Detect says one is IN the
				// gripper, and the two disagree whenever the cap sat crooked or
				// moved as the jaws closed. Lifting on that disagreement carries
				// nothing to the pallet and fits nothing to the part.
				Y_Gripper.Extend();
				IF Y_Gripper.Extended THEN
					IF B_Detect.Active THEN
						SequenceState := SequenceState + 10;
					ELSIF GripTimer.Q THEN
						_FaultCode := 5;
						AbortImmediate();
					END_IF
				END_IF

			80:	// Lift clear before traversing. The next cap comes forward against
				// the held stopper on its own.
				Y_AxisZ2.Retract();
				IF Y_AxisZ2.Retracted THEN
					SequenceState := SequenceState + 10;
				END_IF

			//--- Carry it to the pallet ----------------------------------------
			90:	// Traverse across to the pallet.
				//
				// *** SAFE *** - X max, Z1 min, Z2 min, R min, cap in the gripper. The
				// end of this step IS the safe position, reached in the ordinary course
				// of the cycle rather than only by the reset: both vertical strokes are
				// already up (Z2 at step 80, Z1 untouched), R has not turned yet, and
				// the traverse has just finished. That is why step 100 is the resume
				// entry and why nothing had to be inserted to make the position real -
				// unlike FG_03's arm 1, which never passes through its own safe spot.
				Y_AxisX.Extend();
				IF Y_AxisX.Extended THEN
					SequenceState := SequenceState + 10;
				END_IF

			100: // Rotate into the fitting orientation, in the air and clear of
				// everything
				Y_AxisR.Extend();
				IF Y_AxisR.Extended THEN
					SequenceState := SequenceState + 10;
				END_IF

			110: // Lower onto the part
				Y_AxisZ1.Extend();
				IF Y_AxisZ1.Extended THEN
					SequenceState := SequenceState + 10;
				END_IF

			120: // Release the cap onto the part, and confirm it has left the jaws
				// before the unit lifts. A cap that stays gripped is carried back
				// off the pallet, and the pallet leaves this station uncapped with
				// nothing having reported a problem.
				Y_Gripper.Retract();
				IF Y_Gripper.Retracted THEN
					IF NOT B_Detect.Active THEN
						SequenceState := SequenceState + 10;
					ELSIF ReleaseTimer.Q THEN
						_FaultCode := 6;
						AbortImmediate();
					END_IF
				END_IF

			//--- Return --------------------------------------------------------
			130: // Up, clear of the pallet, before anything traverses
				Y_AxisZ1.Retract();
				IF Y_AxisZ1.Retracted THEN
					SequenceState := SequenceState + 10;
				END_IF

			140: // Back over the feed
				Y_AxisX.Retract();
				IF Y_AxisX.Retracted THEN
					SequenceState := SequenceState + 10;
				END_IF

			150: // Rotate home, ready for the next cap
				Y_AxisR.Retract();
				IF Y_AxisR.Retracted THEN
					SequenceState := SequenceState + 10;
				END_IF

			160: // Execute is the one acting state that does not self-complete.
				// StateComplete() would be wrong here.
				P_Camera.Disable();
				ChangeState(E_PMLCommand.ePMLCommand_Complete);
		END_CASE

	//======================= MAINTENANCE & MANUAL =============================
	E_PMLUnitMode.ePMLUnitMode_Maintenance, E_PMLUnitMode.ePMLUnitMode_Manual:
		// Every device in this group is reachable through its own component HMI
		// struct - the six cylinders through SolenoidHMI, the camera and the
		// bunker through their own. HMIPermissions grants that in these modes and
		// the components honour it themselves. No group sequence runs.
		;
END_CASE

SUPER^.Execute();

SettleTimer(IN := (SequenceState = 10) AND B_Part.Active,	PT := T#500MS);

// One budget from Ready, one from Trigger to verdict. The shot timer spans both
// steps 30 and 40 on purpose: the split between "acknowledged" and "answered" is
// the station's business, but the camera's total response time is one number and
// is what the operator would be told. Same budgets as FG_01 and FG_02 - it is the
// same device.
ReadyTimer(IN := SequenceState = 20,						PT := T#2S);
ShotTimer(IN := (SequenceState = 30) OR (SequenceState = 40),	PT := T#3S);

// The payload grace timers, armed only once the gripper has reached its limit. Same
// budget and same reasoning as FG_03's four: long enough that a slow physics step
// cannot fault a good grip, short enough to be a fault rather than a stall.
GripTimer(IN	:= (SequenceState = 70)  AND Y_Gripper.Extended,		PT := T#500MS);
ReleaseTimer(IN	:= (SequenceState = 120) AND Y_Gripper.Retracted,	PT := T#500MS);
END_METHOD

METHOD PROTECTED HMICommunication
VAR_INPUT
END_VAR
// The command half of the HMI bridge; PublishStatus is the status half.
//
// The base reads its OWN PackMLBaseModule_HMI.Command and never looks at ours, so
// without this a mode or state button on the FG_05 tile writes into a struct
// nothing consumes. It has to happen in this method because the base calls it
// immediately before ModeControl() and StateControl().
PackMLBaseModule_HMI.Command := HMI.Command;

SUPER^.HMICommunication();

// The base clears a latch by writing back the value it acted on, so the panel
// sees its request consumed instead of re-issuing it next scan.
HMI.Command := PackMLBaseModule_HMI.Command;
END_METHOD

METHOD PROTECTED Initialize : BOOL;
VAR
END_VAR
Initialize := FALSE;

CASE DescendantSequenceState OF
	0:
		RegisterComponent(Y_AxisX);
		RegisterComponent(Y_AxisZ1);
		RegisterComponent(Y_AxisZ2);
		RegisterComponent(Y_AxisR);
		RegisterComponent(Y_Gripper);
		RegisterComponent(B_Detect);
		RegisterComponent(Y_CapsSourceStopper);
		RegisterComponent(Y_CapsSource);
		RegisterComponent(B_Part);
		RegisterComponent(P_Camera);

		_LogModeChanges		:= FALSE;
		_LogStateChanges	:= TRUE;
		HMI.Config.Name		:= THIS^._Name;
		DescendantSequenceState := DescendantSequenceState + 10;

	10:
		// Travel timeouts in ms (LREAL). The twin completes a stroke well inside
		// these; they exist to alarm on a jam, not to pace the cycle. The traverse
		// and the rotate are the long strokes.
		Y_AxisX.ExtendTime					:= 3000.0;
		Y_AxisX.RetractTime					:= 3000.0;
		Y_AxisZ1.ExtendTime					:= 2000.0;
		Y_AxisZ1.RetractTime				:= 2000.0;
		Y_AxisZ2.ExtendTime					:= 2000.0;
		Y_AxisZ2.RetractTime				:= 2000.0;
		Y_AxisR.ExtendTime					:= 3000.0;
		Y_AxisR.RetractTime					:= 3000.0;
		Y_Gripper.ExtendTime				:= 2000.0;
		Y_Gripper.RetractTime				:= 2000.0;
		Y_CapsSourceStopper.ExtendTime		:= 2000.0;
		Y_CapsSourceStopper.RetractTime		:= 2000.0;
		DescendantSequenceState := DescendantSequenceState + 10;

	20:
		IF SUPER^.Initialize() THEN
			DescendantSequenceState := DescendantSequenceState + 10;
		END_IF

	30:
		Initialize := TRUE;
END_CASE
END_METHOD

ACTION PublishStatus:
// Local HMI surface, and the status half of the HMI bridge - HMICommunication is
// the command half. Called from CyclicLogic AFTER SUPER^.CyclicLogic(), so every
// field is this scan's. Copy the base struct wholesale - setting fields one by
// one leaves Busy, Error, ErrorID and HMIControlAvailable at zero.
// Every device publishes itself; what is added here is what no device owns.
HMI.Config		:= PackMLBaseModule_HMI.Config;
HMI.Status		:= PackMLBaseModule_HMI.Status;

HMI.StateName				:= F_PMLStateName(_CurrentState);
HMI.Sequence.StepIndex		:= SequenceState;
HMI.Capping.FaultCode		:= _FaultCode;
HMI.Capping.LastResultOK	:= _LastResultOK;

// ResumePoint IS DERIVED HERE, NOT COPIED FROM _Held. That one is Resetting's
// private snapshot and is stale everywhere else. This runs the same derivation
// Execute step 0 runs, off the live sensor, so the panel shows what pressing Start
// would actually do rather than what the last reset happened to see.
IF B_Detect.Active THEN
	HMI.Capping.ResumePoint := 2;		// place the cap already held
ELSE
	HMI.Capping.ResumePoint := 1;		// the whole cycle
END_IF
END_ACTION

METHOD PROTECTED Resetting
VAR_INPUT
END_VAR
// Home the cap handling unit from wherever the cycle stopped.
// THE ORDER IS THE COLLISION ANALYSIS. Both vertical strokes come up first, which
// is always safe; only then does anything traverse or rotate, which with the
// gripper high is also safe. Any other order can drag a lowered gripper across the
// pallet or into the feed conveyor.
//
// Every step waits on its own cylinders and nothing else - not B_Part, not
// B_Detect, not the index unit. B_Detect is SAMPLED ONCE at step 0 and never read
// again: a snapshot selects the ending, a live read could stall it.
//
// THE RESET KEEPS THE CAP AND PARKS IT AT THE SAFE POSITION:
//   SAFE   X MAX, Z1 min, Z2 min, R min, cap in the gripper
// which is exactly what Execute step 90 leaves, so the cycle resumes at step 100.
//
// The alternatives are all wrong, and it is worth recording why:
//   Back on the feed?  The pick position is not empty - the next cap advanced
//                      against the held stopper. Two caps on one position jams it.
//   Onto the part?     A reset does not deliver product, and it would mean knowing
//                      Index05 still has a pallet clamped - waiting on another unit.
//   Open in the air?   The cap falls.
//   Keep it and stop?  Turns every E-Stop into a trip into the cell for a cap that
//                      was never in danger.

CASE SequenceState OF
	0:
		// BLOCK THE FEED BEFORE ANYTHING HOMES. The stopper's de-energised position no
		// longer blocks the path - EXTENDED does, since the device was refactored in
		// the twin - and DriveBunker keeps the feed running right through Resetting and
		// Idle. Commanded here rather than at step 30, the queue accumulates against the
		// stopper from the first scan of the reset instead of spilling past the pick
		// position while the axes home. The command latches, so step 30 only has to
		// wait on .Extended and the state still terminates on this unit's own travel
		// budget.
		NoStateTasksToComplete	:= FALSE;
		Y_CapsSourceStopper.Extend();
		P_Camera.Disable();
		_Held					:= B_Detect.Active;
		SequenceState			:= SequenceState + 10;

	10:	// Both vertical strokes up. Commanded on the same scan so they travel
		// together rather than one after the other.
		Y_AxisZ1.Retract();
		Y_AxisZ2.Retract();
		IF Y_AxisZ1.Retracted AND Y_AxisZ2.Retracted THEN
			SequenceState := SequenceState + 10;
		END_IF

	20:	// Rotate home, and traverse to whichever end of X this unit can stand at.
		// R always goes home: it is min at the safe position and min at rest, so
		// there is nothing to decide. X is the one that depends on the payload -
		// MAX with a cap, which is the pallet side and the safe position, min
		// without one, which is the feed side and home.
		//
		// Both vertical strokes are up from step 10, so the unit can cross freely
		// in either direction and turn while it does.
		Y_AxisR.Retract();

		IF _Held THEN
			Y_AxisX.Extend();
			IF Y_AxisX.Extended AND Y_AxisR.Retracted THEN
				SequenceState := SequenceState + 10;
			END_IF
		ELSE
			Y_AxisX.Retract();
			IF Y_AxisX.Retracted AND Y_AxisR.Retracted THEN
				SequenceState := SequenceState + 10;
			END_IF
		END_IF

	30:	// Confirm the feed is blocked - the stopper was commanded at step 0 - and
		// open the gripper only if it is empty.
		//
		// With a cap held, Y_Gripper is not commanded HERE - CyclicLogic is holding
		// it closed instead, and that command wins because it runs first. The step
		// then waits on the stopper alone, which is still this unit's own cylinder,
		// so the state still terminates on its own travel budget. No fault is
		// raised: a cap parked at the safe position is a resumable cycle, not a
		// problem.
		Y_CapsSourceStopper.Extend();

		IF _Held THEN
			IF Y_CapsSourceStopper.Extended THEN
				SequenceState := SequenceState + 10;
			END_IF
		ELSE
			Y_Gripper.Retract();
			IF Y_Gripper.Retracted AND Y_CapsSourceStopper.Extended THEN
				SequenceState := SequenceState + 10;
			END_IF
		END_IF

	40:
		StateTasksComplete := TRUE;
END_CASE

SUPER^.Resetting();
END_METHOD

METHOD PROTECTED Stopping
VAR_INPUT
END_VAR
// A controlled stop commands no axis motion, for the same reason the abort does
// not: a cap is held in the air for most of this cycle, and the grip is held by the
// CyclicLogic interlock rather than by leaving the valve alone. The feed and the
// camera stop, because both run on their own and neither should keep running into a
// stopped station.
CASE SequenceState OF
	0:
		NoStateTasksToComplete	:= FALSE;
		Y_CapsSource.Halt();
		P_Camera.Disable();
		SequenceState			:= SequenceState + 10;

	10:
		StateTasksComplete := TRUE;
END_CASE

SUPER^.Stopping();
END_METHOD

END_FUNCTION_BLOCK

// ---- Library/POUs/FB_AbstractBunker.TcPOU
// Generic byte-oriented parts bunker component.
// Bit layout, from the twin node MAIN.FG_05.Y_CapsSource:
//   Output: 0 vibration table, 1 feed conveyor.   Input: unused.
//
// AN OUTPUT-ONLY DEVICE. No feedback, so nothing to time out on: _Busy and _Error
// stay false and the status struct mirrors the commanded bits. A travel timeout or
// a "table stalled" fault would be a fiction, and a plausible fiction gets believed.
//
// Not part of any pallet cycle - the feed runs continuously so caps accumulate at
// the pick position between pallets. FG_05 drives it from CyclicLogic, never Execute.
FUNCTION_BLOCK FB_AbstractBunker EXTENDS FB_ComponentBase
VAR
	// Declared and linked though the twin drives nothing into it: the twin device
	// is an FB_DeviceByte and carries the pair whatever this side does, so the
	// channel exists. Nothing in this block consumes it.
	InputData  AT %I* : BYTE;
	OutputData AT %Q* : BYTE;
	{ attribute 'TcHmiSymbol.AddSymbol' }
	HMI : ST_AbstractBunker_HMI;
END_VAR

METHOD PUBLIC CyclicLogic
VAR_INPUT END_VAR
IF NOT _InitComplete THEN
	_InitComplete := Initialize();
	RETURN;
END_IF

SUPER^.CyclicLogic();

// Commanded state, not measured state - see the block header.
HMI.Device.TableRunning		:= OutputData.0;
HMI.Device.ConveyorRunning	:= OutputData.1;
END_METHOD

// Table first: stopping the conveyor while the table still feeds it piles caps up
// at the transfer point.
METHOD PUBLIC Halt
VAR_INPUT END_VAR
OutputData.0 := FALSE;
OutputData.1 := FALSE;
END_METHOD

METHOD PROTECTED HMICommunication
VAR_INPUT END_VAR
// HMI is a published mirror of the base's own ComponentBase_HMI - carry operator
// intent in before the base looks, and its answers back out afterwards.
ComponentBase_HMI.Command := HMI.Command;

SUPER^.HMICommunication();

HMI.Config	:= ComponentBase_HMI.Config;
HMI.Status	:= ComponentBase_HMI.Status;
HMI.Command	:= ComponentBase_HMI.Command;

IF ComponentBase_HMI.Status.HMIControlAvailable THEN
	OutputData.0 := HMI.DeviceCommand.RunTable;
	OutputData.1 := HMI.DeviceCommand.RunConveyor;
ELSE
	HMI.DeviceCommand.RunTable		:= OutputData.0;
	HMI.DeviceCommand.RunConveyor	:= OutputData.1;
END_IF
END_METHOD

METHOD PROTECTED Initialize : BOOL
VAR_INPUT END_VAR
Initialize := SUPER^.Initialize();
END_METHOD

// Conveyor first, so the pick position is being cleared before the table starts
// feeding into it.
METHOD PUBLIC Run
VAR_INPUT END_VAR
OutputData.1 := TRUE;
OutputData.0 := TRUE;
END_METHOD

// TRUE when both halves of the feed are commanded on. Commanded, not confirmed -
// this device has no status byte.
PROPERTY Running : BOOL
GET
Running := OutputData.0 AND OutputData.1;
END_GET
END_PROPERTY

END_FUNCTION_BLOCK

// ---- Library/POUs/FB_ControlSource_HMI.TcPOU
// ============================================================================
// Connects the TwinCAT HMI to the machine's PackML state machine.
// The HMI binds straight to the inherited structs - FB_ControlSource already
// exposes the right shape in the standard PackML types
// (MainPMLControl_Standard.CurrentState/CurrentMode/StateCommand/ModeCommand,
// MainPMLControl_Simplified.*Permissive). The base refreshes the actuals,
// recomputes the permissives and acts on a changed command; all this block adds is
// the command latch release below.
// Registered by MAIN via Machine.RegisterExternalController(THIS^).
{ attribute 'TcHmiSymbol.AddSymbol' }
FUNCTION_BLOCK FB_ControlSource_HMI EXTENDS FB_ControlSource
VAR
END_VAR

METHOD PUBLIC CyclicLogic
VAR_INPUT
END_VAR
// Until RegisterExternalController has run, the base has no module to talk to
// and its CyclicLogic would dereference a null interface.
IF NOT Registered THEN
	RETURN;
END_IF

SUPER^.CyclicLogic();

ReleaseCommandLatch();
END_METHOD

ACTION ReleaseCommandLatch:
// The base treats a command as "StateCommand differs from StateCommandLast", and
// stamps StateCommandLast once it has acted, so pressing the same button twice in
// a row would be swallowed the second time. Clearing both together, after the base
// has acted, makes every press count.
// ModeCommand is deliberately NOT cleared - selecting the same mode twice is a
// no-op anyway.
IF MainPMLControl_Standard.StateCommand <> E_PMLCommand.ePMLCommand_Undefined THEN
	MainPMLControl_Standard.StateCommand		:= E_PMLCommand.ePMLCommand_Undefined;
	MainPMLControl_Standard.StateCommandLast	:= E_PMLCommand.ePMLCommand_Undefined;
END_IF
END_ACTION

END_FUNCTION_BLOCK

// ---- Library/POUs/FB_ControlSource_Panel.TcPOU
// ============================================================================
// The physical operator panel, H_ControlPanel, as a PackML control source.
//
// WHY A CONTROL SOURCE AND NOT A DEVICE. FB_ControlSource already contains the
// whole START/STOP/RESET ladder, and ST_PackML_Control_Simplified declares its
// three *Pressed members AT %I* - so three of the eight buttons need no code at
// all: they are linked in Mapping_PLC.xml. Only the other five are translated here.
//
// Twin bit layout, verified 2026-08-20 against the live PanelSampler:
//   StatusData bit0 START  bit1 RESET  bit2 STOP    bit3 CLEAR
//              bit4 ABORT  bit5 PRODUCTION  bit6 MAINTANANCE  bit7 MANUAL
//   ControlData carries each button's own lamp at the same bit.
//
// DELIBERATE DEVIATION: the SPT library says Abort "should not be directly
// commanded from any user inteface". This panel does exactly that - chosen
// knowingly by the project owner over routing the button into the safety chain.
FUNCTION_BLOCK FB_ControlSource_Panel EXTENDS FB_ControlSource
VAR
	// The five buttons the base does not handle. START / STOP / RESET are the
	// inherited MainPMLControl_Simplified.*Pressed members and are linked there.
	ClearPressed AT %I* : BOOL;
	AbortPressed AT %I* : BOOL;
	ProductionPressed AT %I* : BOOL;
	MaintenancePressed AT %I* : BOOL;
	ManualPressed AT %I* : BOOL;

	// Button lamps, ControlData bits 0..7 in panel order.
	LampStart AT %Q* : BOOL;
	LampReset AT %Q* : BOOL;
	LampStop AT %Q* : BOOL;
	LampClear AT %Q* : BOOL;
	LampAbort AT %Q* : BOOL;
	LampProduction AT %Q* : BOOL;
	LampMaintenance AT %Q* : BOOL;
	LampManual AT %Q* : BOOL;

	// Written by MAIN each scan.
	_Flash : BOOL;		// shared flash phase, from the signal tower
	_SafetyOk : BOOL;	// the machine's derived safety chain

	ButtonTrigger : R_TRIG;

	StartFlash : BOOL;
	StartSolid : BOOL;
	ResetFlash : BOOL;
END_VAR

METHOD PUBLIC CyclicLogic
VAR_INPUT
END_VAR
// Until RegisterExternalController has run, the base has no module to talk to
// and its CyclicLogic would dereference a null interface.
IF NOT Registered THEN
	RETURN;
END_IF

// Before SUPER^: the base's command R_TRIG folds StateCommand / ModeCommand
// changes into its clock, so a command written now is acted on this scan.
TranslateButtons();

SUPER^.CyclicLogic();

ReleaseCommandLatch();

// AFTER SUPER^, which has just recomputed the permissives. Vetoing them here gates
// the NEXT scan's command ladder, and keeps the lamps honest - a vetoed button
// stays dark instead of inviting a press that would do nothing.
IF NOT _SafetyOk THEN
	MainPMLControl_Simplified.StartPermissive := FALSE;
	MainPMLControl_Simplified.ResetPermissive := FALSE;
END_IF

DriveLamps();
END_METHOD

ACTION DriveLamps:
// The three rows of state-lamp.md that name a button, plus five lamps the table
// says nothing about. The latter are a project choice and are marked as such.

// --- Ready to Start -> Start Button Flashing --------------------------------
// The table says Idle only. StartPermissive is Idle OR Held, so both are tested:
// the lamp then reflects what a press would actually do.
StartFlash := (MainPMLControl_Standard.CurrentState = Tc3_PackML_V2.E_PMLState.ePMLState_Idle)
			AND MainPMLControl_Simplified.StartPermissive;

// --- Running -> Start Button Solid ------------------------------------------
// NOTE this row is NOT the same set as the green lamp's Running row: the button
// stays solid through Suspending and Suspended, the tower's green does not.
StartSolid :=	(MainPMLControl_Standard.CurrentState = Tc3_PackML_V2.E_PMLState.ePMLState_Starting)
			OR	(MainPMLControl_Standard.CurrentState = Tc3_PackML_V2.E_PMLState.ePMLState_Execute)
			OR	(MainPMLControl_Standard.CurrentState = Tc3_PackML_V2.E_PMLState.ePMLState_Completing)
			OR	(MainPMLControl_Standard.CurrentState = Tc3_PackML_V2.E_PMLState.ePMLState_Unholding)
			OR	(MainPMLControl_Standard.CurrentState = Tc3_PackML_V2.E_PMLState.ePMLState_Suspending)
			OR	(MainPMLControl_Standard.CurrentState = Tc3_PackML_V2.E_PMLState.ePMLState_Suspended)
			OR	(MainPMLControl_Standard.CurrentState = Tc3_PackML_V2.E_PMLState.ePMLState_Unsuspending);

// --- Ready to Reset -> Reset Button Flashing --------------------------------
// Aborted, Complete and Stopped - which is exactly ResetPermissive, so the
// vetoed permissive alone carries it.
ResetFlash := MainPMLControl_Simplified.ResetPermissive;

LampStart	:= (StartFlash AND _Flash) OR StartSolid;
LampReset	:= ResetFlash AND _Flash;

// --- Beyond the table -------------------------------------------------------
// state-lamp.md does not cover these five. Solid-when-actionable for the command
// buttons, solid-on-active for the mode buttons.
LampStop	:= MainPMLControl_Simplified.StopPermissive;
LampClear	:= (MainPMLControl_Standard.CurrentState = Tc3_PackML_V2.E_PMLState.ePMLState_Aborted);
LampAbort	:= ((MainPMLControl_Standard.CurrentState = Tc3_PackML_V2.E_PMLState.ePMLState_Aborting)
			 OR		(MainPMLControl_Standard.CurrentState = Tc3_PackML_V2.E_PMLState.ePMLState_Aborted)
			 OR		(MainPMLControl_Standard.CurrentState = Tc3_PackML_V2.E_PMLState.ePMLState_Clearing));

LampProduction		:= (MainPMLControl_Standard.CurrentMode = E_PMLUnitMode.ePMLUnitMode_Production);
LampMaintenance	:= (MainPMLControl_Standard.CurrentMode = E_PMLUnitMode.ePMLUnitMode_Maintenance);
LampManual			:= (MainPMLControl_Standard.CurrentMode = E_PMLUnitMode.ePMLUnitMode_Manual);
END_ACTION

// Shared flash phase, taken from the signal tower so every flashing lamp on the
// machine blinks together.
PROPERTY Flash : BOOL
GET
Flash := _Flash;
END_GET
SET
_Flash := Flash;
END_SET
END_PROPERTY

ACTION ReleaseCommandLatch:
// Identical to FB_ControlSource_HMI's latch release, and needed for the same
// reason: the base stamps StateCommandLast once it has acted, so the same button
// pressed twice would be swallowed. ModeCommand is deliberately NOT cleared.
IF MainPMLControl_Standard.StateCommand <> E_PMLCommand.ePMLCommand_Undefined THEN
	MainPMLControl_Standard.StateCommand		:= E_PMLCommand.ePMLCommand_Undefined;
	MainPMLControl_Standard.StateCommandLast	:= E_PMLCommand.ePMLCommand_Undefined;
END_IF
END_ACTION

// The machine's derived safety chain, written by MAIN each scan. FALSE vetoes
// the Start and Reset permissives.
PROPERTY SafetyOk : BOOL
GET
SafetyOk := _SafetyOk;
END_GET
SET
_SafetyOk := SafetyOk;
END_SET
END_PROPERTY

ACTION TranslateButtons:
// One edge across all five, then priority order. Two buttons pressed on the same
// scan resolve by the ELSIF chain rather than fighting.
ButtonTrigger(CLK :=	ClearPressed
					OR	AbortPressed
					OR	ProductionPressed
					OR	MaintenancePressed
					OR	ManualPressed);

IF ButtonTrigger.Q THEN
	IF AbortPressed THEN
		// See the deviation note in the declaration header.
		MainPMLControl_Standard.StateCommand := E_PMLCommand.ePMLCommand_Abort;

	ELSIF ClearPressed THEN
		MainPMLControl_Standard.StateCommand := E_PMLCommand.ePMLCommand_Clear;

	ELSIF ProductionPressed THEN
		MainPMLControl_Standard.ModeCommand := E_PMLUnitMode.ePMLUnitMode_Production;

	ELSIF MaintenancePressed THEN
		MainPMLControl_Standard.ModeCommand := E_PMLUnitMode.ePMLUnitMode_Maintenance;

	ELSIF ManualPressed THEN
		MainPMLControl_Standard.ModeCommand := E_PMLUnitMode.ePMLUnitMode_Manual;
	END_IF
END_IF
END_ACTION

END_FUNCTION_BLOCK
